{attribute 'qualified_only'}
{attribute 'strict'}
TYPE E_Mode :
(
	Segment := 1,
	Level	:= 2,
	Runlight:= 4
);
END_TYPE

(* stored: Version 1.1.0.1, ProductVersion 3.1.4024.10
   DUT E_Mode: Id {37b4b9bc-fb7d-4473-8c4f-cb81c8bc6a9f} *)
